{attribute 'qualified_only'}
{attribute 'strict'}
TYPE E_MachineState :
(
	IDLE := 0,
	Drilling,
	Retracting,
	Error
);
END_TYPE

(* stored: Version 1.1.0.1, ProductVersion 3.1.4024.16
   DUT E_MachineState: Id {a48a40ce-d553-4c7d-8d50-972c72329fd0} *)
